FUNCTION_BLOCK JsonDecoderTest EXTENDS JsonDecoder IMPLEMENTS IUnitTest

METHOD Test_Decode_NestedArray
VAR_INPUT
  assertions : IAssertions;
END_VAR
VAR
  element0 : IJsonElement;
  element1 : IJsonElement;
  element2 : IJsonElement;  
END_VAR
Decode('[[[4,2,3]]]');
element0 := Element('array[0][0][0]');
element1 := Element('array[0][0][1]');
element2 := Element('array[0][0][2]');

assertions.IsTrue(element0 <> 0, '');
assertions.IsTrue(element1 <> 0, '');
assertions.IsTrue(element2 <> 0, '');

IF element0 <> 0 AND element1 <> 0 AND element2 <> 0
THEN
	assertions.EqualsString('4', element0.AsString(), '');
	assertions.EqualsString('2', element1.AsString(), '');
	assertions.EqualsString('3', element2.AsString(), '');
END_IF
END_METHOD

METHOD Test_IntToString
VAR_INPUT
  assertions : IAssertions;
END_VAR
VAR
  str : STRING;
END_VAR
str := '';
IntToString(0, str);
assertions.EqualsString(expected := '0', actual := str, message:='Index 0 is correctly converted to an array index key');

str := '';
IntToString(1, str);
assertions.EqualsString(expected := '1', actual := str, message:='Index 1 is correctly converted to an array index key');

str := '';
IntToString(9, str);
assertions.EqualsString(expected := '9', actual := str, message:='Index 9 is correctly converted to an array index key');

str := '';
IntToString(10, str);
assertions.EqualsString(expected := '10', actual := str, message:='Index 10 is correctly converted to an array index key');

str := '';
IntToString(55, str);
assertions.EqualsString(expected := '55', actual := str, message:='Index 55 is correctly converted to an array index key');
END_METHOD

METHOD Test_SkipWhitespace
VAR_INPUT
  assertions : IAssertions;
END_VAR
VAR
  json : STRING;  
END_VAR
json := '              

        !';
_jsonPtr := ADR(json);
SkipWhitespaces();

_jsonPtr^ := 16#33;
END_METHOD

END_FUNCTION_BLOCK

(* stored: Version 1.1.0.1, ProductVersion 3.1.4024.12
   POU JsonDecoderTest: Id {f5f16609-da6a-435e-8d26-a4efca0c555c}, SpecialFunc None
   Method Test_Decode_NestedArray: Id {8270d688-a825-4732-8ad8-272f25321512}
   Method Test_IntToString: Id {997eece4-29aa-4921-82a5-00c9de6877a1}
   Method Test_SkipWhitespace: Id {dc82c6e9-cadf-4c97-bb57-c8902c8d6d57} *)
